// TIA Portal project "Traffic Barrier Control" (V17)
// Traffic Barrier Control
// When a vehicle arrives, raise the barrier for 20 sec and after that lower the barrier.
// If the barrier hits during lowering, immediately stop and raise the barrier for 5 sec again.

(* hardware
DEVICE "S7-1200 station_1"  S7-1200 Station
   slot 0: "Rack_0"  S7-1200 Rack  Rack  V1.0
   slot 1: "PLC_1"  CPU 1212C AC/DC/Rly  6ES7 212-1BE40-0XB0  V4.5
*)

// ===== PLC "PLC_1"  CPU 1212C AC/DC/Rly =====

VAR_GLOBAL   // PLC tag table "Default tag table"
   "Sensor" AT %I0.0 : Bool;
   "Barrier" AT %Q0.0 : Bool;
   "Tag_1" AT %M0.0 : Bool;
   "Tag_2" AT %M0.1 : Bool;
   "Tag_3" AT %M0.2 : Bool;
END_VAR

// folder: System blocks/Program resources

DATA_BLOCK "IEC_Timer_0_DB"   // DB1
{ S7_Optimized_Access := 'TRUE' }
AUTHOR : Simatic
FAMILY : IEC
NAME : IEC_TMR
VERSION : 1.0
// stored: InstanceOfName IEC_TIMER
"IEC_TIMER"
BEGIN
END_DATA_BLOCK

DATA_BLOCK "IEC_Timer_0_DB_1"   // DB2
{ S7_Optimized_Access := 'TRUE' }
AUTHOR : Simatic
FAMILY : IEC
NAME : IEC_TMR
VERSION : 1.0
// stored: InstanceOfName IEC_TIMER
"IEC_TIMER"
BEGIN
END_DATA_BLOCK

DATA_BLOCK "IEC_Timer_0_DB_2"   // DB3
{ S7_Optimized_Access := 'TRUE' }
AUTHOR : Simatic
FAMILY : IEC
NAME : IEC_TMR
VERSION : 1.0
// stored: InstanceOfName IEC_TIMER
"IEC_TIMER"
BEGIN
END_DATA_BLOCK

// folder: (top level)

ORGANIZATION_BLOCK "Main"   // OB1, LAD, ProgramCycle
TITLE = "Main Program Sweep (Cycle)"
{ S7_Optimized_Access := 'TRUE' }
VERSION : 0.1
   VAR_INPUT
      Initial_Call : Bool;   // Initial call of this OB
      Remanence : Bool;   // =True, if remanent data are available
   END_VAR
BEGIN

REGION Network 1
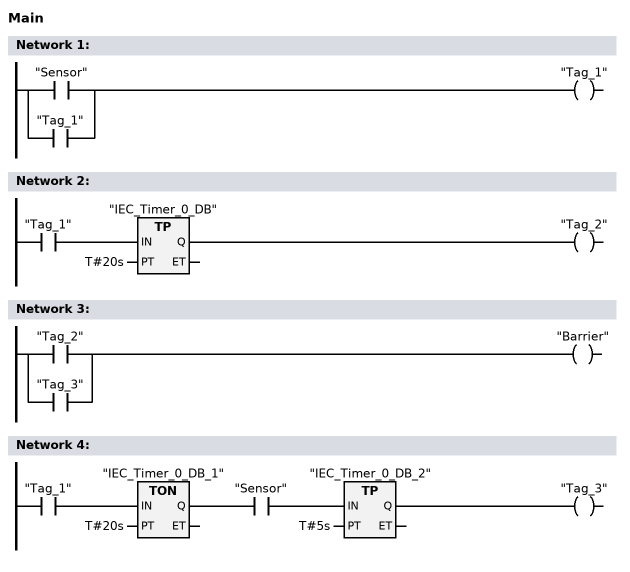
   RUNG wire#powerrail
      Contact( "Sensor" )
      wire#w1
      Coil( "Tag_1" )
   END_RUNG
   RUNG wire#powerrail
      Contact( "Tag_1" )
   END_RUNG wire#w1
   // the same network as SCL:
   "Tag_1" := "Sensor" OR "Tag_1";
END_REGION

REGION Network 2
   "IEC_Timer_0_DB".TP(IN := "Tag_1", PT := T#20s);
   "Tag_2" := "IEC_Timer_0_DB".Q;
END_REGION

REGION Network 3
   RUNG wire#powerrail
      Contact( "Tag_2" )
      wire#w1
      Coil( "Barrier" )
   END_RUNG
   RUNG wire#powerrail
      Contact( "Tag_3" )
   END_RUNG wire#w1
   // the same network as SCL:
   "Barrier" := "Tag_2" OR "Tag_3";
END_REGION

REGION Network 4
   "IEC_Timer_0_DB_1".TON(IN := "Tag_1", PT := T#20s);
   "IEC_Timer_0_DB_2".TP(IN := "IEC_Timer_0_DB_1".Q AND "Sensor", PT := T#5s);
   "Tag_3" := "IEC_Timer_0_DB_2".Q;
END_REGION
END_ORGANIZATION_BLOCK